DATA_BLOCK "A-DBVALVES"
TITLE = DBVALVES
{ S7_Optimized_Access := 'TRUE' }
AUTHOR : PiotrSlezak
FAMILY : Vorster
VERSION : 0.2
NON_RETAIN
//Blok danych stanowiący interface obsługi, diagnostyki i wizualizacji elektrozaworów i siłowników
   VAR
      LAMP_TEST { S7_SetPoint := 'False'} : Bool;
BR : Struct
	PIN_RISING_01 { S7_SetPoint := 'False'} : "Tstate";   // [5] BR pin_podnoszenie_01
	PIN_01 { S7_SetPoint := 'False'} : "Tstate";   // [6] BR pin_01
	PIN_RISING_02 { S7_SetPoint := 'False'} : "Tstate";   // [7] BR pin_podnoszenie_02
	PIN_02 { S7_SetPoint := 'False'} : "Tstate";   // [8] BR pin_02
	PIN_RISING_03 { S7_SetPoint := 'False'} : "Tstate";   // [9] BR pin_podnoszenie_03
	PIN_03 { S7_SetPoint := 'False'} : "Tstate";   // [10] BR pin_03
	PIN_RISING_04 { S7_SetPoint := 'False'} : "Tstate";   // [11] BR pin_podnoszenie_04
	PIN_04 { S7_SetPoint := 'False'} : "Tstate";   // [12] BR pin_04
	TABLE5_FRONT { S7_SetPoint := 'False'} : "Tstate";   // [13] BR blat5_przod
	TABLE_REAR_LEFT { S7_SetPoint := 'False'} : "Tstate";   // [14] BR blat_tyl_lewy
	TABLE_REAR_RIGHT { S7_SetPoint := 'False'} : "Tstate";   // [15] BR blat_tyl_prawy
END_STRUCT;
GN : Struct
	SCREW_LOCK_LEFT { S7_SetPoint := 'False'} : "Tstate";   // [1] GN blokada_sruby_lewy
	SCREW_LOCK_MIDDLE { S7_SetPoint := 'False'} : "Tstate";   // [2] GN blokada_sruby_srodek
	SCREW_LOCK_RIGHT { S7_SetPoint := 'False'} : "Tstate";   // [3] GN blokada_sruby_prawy
	LATCH { S7_SetPoint := 'False'} : "Tstate";   // [4] GN zasuwka
END_STRUCT;
ST1 : Struct
	STATION_MOVEMENT { S7_SetPoint := 'False'} : "Tstate";   // [16] ST1 przesuw_stacji
	SWORD_SLIDE_OUT { S7_SetPoint := 'False'} : "Tstate";   // [17] ST1 wysuw_miecza
	SWORD { S7_SetPoint := 'False'} : "Tstate";   // [18] ST1 miecz
END_STRUCT;
ST2 : Struct
	STATION_MOVEMENT { S7_SetPoint := 'False'} : "Tstate";   // [19] ST2 przesuw_stacji
	SWORD_SLIDE_OUT { S7_SetPoint := 'False'} : "Tstate";   // [20] ST2 wysuw_miecza
	SWORD { S7_SetPoint := 'False'} : "Tstate";   // [21] ST2 miecz
END_STRUCT;
ST3 : Struct
	SWORD { S7_SetPoint := 'False'} : "Tstate";   // [22] ST3 miecz
	BUMPER { S7_SetPoint := 'False'} : "Tstate";   // [23] ST3 zderzak
	SWORD_RISING { S7_SetPoint := 'False'} : "Tstate";   // [24] ST3 podnoszenie_miecza
END_STRUCT;
ST4 : Struct
	SWORD { S7_SetPoint := 'False'} : "Tstate";   // [25] ST4 miecz
	BUMPER { S7_SetPoint := 'False'} : "Tstate";   // [26] ST4 zderzak
	SWORD_RISING { S7_SetPoint := 'False'} : "Tstate";   // [27] ST4 podnoszenie_miecza
END_STRUCT;
ST5 : Struct
	STATION_MOVEMENT { S7_SetPoint := 'False'} : "Tstate";   // [28] ST5 przesuw_stacji
	STATION_SMALL_STEP { S7_SetPoint := 'False'} : "Tstate";   // [29] ST5 stacja_maly_skok
	STATION_BIG_STEP { S7_SetPoint := 'False'} : "Tstate";   // [30] ST5 stacja_duzy_skok
	PIN { S7_SetPoint := 'False'} : "Tstate";   // [31] ST5 pin
END_STRUCT;
ST6 : Struct
	STATION_MOVEMENT { S7_SetPoint := 'False'} : "Tstate";   // [32] ST6 przesuw_stacji
	STATION_SMALL_STEP { S7_SetPoint := 'False'} : "Tstate";   // [33] ST6 stacja_maly_skok
	STATION_BIG_STEP { S7_SetPoint := 'False'} : "Tstate";   // [34] ST6 stacja_duzy_skok
	PIN { S7_SetPoint := 'False'} : "Tstate";   // [35] ST6 pin
END_STRUCT;
ST7 : Struct
	SWORD_1L_MOVEMENT { S7_SetPoint := 'False'} : "Tstate";   // [36] ST7 przesuw_miecza_1l
	SWORD_1R_MOVEMENT { S7_SetPoint := 'False'} : "Tstate";   // [37] ST7 przesuw_miecza_1p
	HOLDFAST_MOVEMENT { S7_SetPoint := 'False'} : "Tstate";   // [38] ST7 przesuw_dociskow
	SWORD_Y_2L_MOVEMENT { S7_SetPoint := 'False'} : "Tstate";   // [39] ST7 przesuw_miecza_y_2l
	SWORD_2L { S7_SetPoint := 'False'} : "Tstate";   // [40] ST7 miecz_2l
	SWORD_Y_2R_MOVEMENT { S7_SetPoint := 'False'} : "Tstate";   // [41] ST7 przesuw_miecza_y_2p
	SWORD_2R { S7_SetPoint := 'False'} : "Tstate";   // [42] ST7 miecz_2p
	SWORD_X_3L_MOVEMENT { S7_SetPoint := 'False'} : "Tstate";   // [43] ST7 przesuw_miecza_x_3l
	SWORD_Y_3L_MOVEMENT { S7_SetPoint := 'False'} : "Tstate";   // [44] ST7 przesuw_miecza_y_3l
	SWORD_3L { S7_SetPoint := 'False'} : "Tstate";   // [45] ST7 miecz_3l
	SWORD_X_3R_MOVEMENT { S7_SetPoint := 'False'} : "Tstate";   // [46] ST7 przesuw_miecza_x_3p
	SWORD_Y_3R_MOVEMENT { S7_SetPoint := 'False'} : "Tstate";   // [47] ST7 przesuw_miecza_y_3p
	SWORD_3R { S7_SetPoint := 'False'} : "Tstate";   // [48] ST7 miecz_3p
	COMB_SLIDE_OUT { S7_SetPoint := 'False'} : "Tstate";   // [49] ST7 wysuw_grzebienia
	COMB { S7_SetPoint := 'False'} : "Tstate";   // [50] ST7 grzebien
END_STRUCT;

   io : Array[0..50] of "Tio";
   END_VAR


BEGIN

END_DATA_BLOCK

